// TIA Portal V19 export
DATA_BLOCK "FinalCutLub"   // DB219
{ DB_Accessible_From_OPC_UA := 'FALSE' }
// stored: DBAccessibleFromOPCUA false, InstanceOfName DiesLubrication_FB, InstanceOfType FB
"DiesLubrication_FB"
   // VAR_INPUT
   //    AreaInterface : "AreaInterface";
   //    DataIn : Struct
   //       PbStop : Bool;
   //       PbStart : Bool;
   //       SensorLevel : Bool;
   //       ConnectorPlugged : Bool;
   //    END_STRUCT;
   //    CIn : Struct
   //       EnableStopInPhase : Bool;
   //       EnableStopProgrammed : Bool;
   //       EnableAborting : Bool;
   //       JobDone : Bool;
   //       ExternalPumpCycleDone : Bool;
   //       CutBenchCode : DInt;
   //    END_STRUCT;
   //    Config : Struct
   //       EnableWngSystemOff : Bool;
   //       ExternalPump : Bool;
   //       PumpWorkDuration : Time;
   //       PumpPauseDuration : Time;
   //       LowTankLevelDly : Time;
   //    END_STRUCT;
   // END_VAR
   // VAR_OUTPUT
   //    MachineInterface : "MachineInterface";
   //    DataOut : Struct
   //       PneumaticPumpSolenoidValve : Bool;
   //       Lamp : Bool;
   //    END_STRUCT;
   //    COut : Struct
   //       IsRunning : Bool;
   //       ToolsJobCounter : UDInt;
   //       PumpCycleCounter : UDInt;
   //    END_STRUCT;
   // END_VAR
   // VAR_IN_OUT
   //    PersistentValues : Struct
   //       Data : Struct
   //          SavedCutBenchCode : DInt;
   //          PumpJobCounter : UDInt;
   //          JobsCounter : UDInt;
   //       END_STRUCT;
   //       Par : Struct
   //          SystemOffOn : Bool;
   //          JobsToStart : UDInt;
   //          OilPumpCycles : UDInt;
   //       END_STRUCT;
   //    END_STRUCT;
   // END_VAR
   // VAR
   //    Sts : Struct
   //       AlarmsPresence : Bool;
   //       WarningsPresence : Bool;
   //       IsStandstill : Bool;
   //       PumpPauseDone : Bool;
   //       PumpWorkDone : Bool;
   //       LubNormCycleReq : Bool;
   //       Condition { ExternalAccessible := 'False'; ExternalVisible := 'False'; ExternalWritable := 'False'} : Bool;
   //    END_STRUCT;
   //    Ctrl : Struct
   //       RstAlarms : Bool;
   //       SafeMotion : Bool;
   //       StopDoorOpen : Bool;
   //       StopSafe : Bool;
   //       StopInPhase : Bool;
   //       StopProgrammed : Bool;
   //       ManStart : Bool;
   //       AutStart : Bool;
   //       V_Pneumatic : Bool;
   //    END_STRUCT;
   //    Warning : Struct
   //       NoAutReady : Bool;
   //       SystemOff : Bool;
   //    END_STRUCT;
   //    Alarm : Struct
   //       LowTankLevel : Bool;
   //       ConnectorUnplugged : Bool;
   //    END_STRUCT;
   //    TON_PumpPause : IEC_TIMER;
   //    TON_PumpWork : IEC_TIMER;
   //    TON_LowTankLevel : IEC_TIMER;
   //    JobDonePEAux : Bool;
   //    PbStartPEAux : Bool;
   // END_VAR
BEGIN
END_DATA_BLOCK
